Staubli VAL3: recvHeartbeat.pgx

public program recvHeartbeat()
  local num l_nByte
  local num l_nBytesRecv
  local num l_nHtbt
  local num l_nHtbtB[4]
  local num l_nIndex
begin
  // Copyright (c) 2016, Ocado Technology - Robotics Research Team
  //
  // Licensed under the Apache License, Version 2.0 (the "License");
  // you may not use this file except in compliance with the License.
  // You may obtain a copy of the License at
  //
  //     http://www.apache.org/licenses/LICENSE-2.0
  //
  // Unless required by applicable law or agreed to in writing, software
  // distributed under the License is distributed on an "AS IS" BASIS,
  // WITHOUT WARRANTIES OR CONDITIONS OF ANY KIND, either express or implied.
  // See the License for the specific language governing permissions and
  // limitations under the License.

nOutConnFlag = 1

end
